P[3275]{
   GP1:
	UF : 7, UT : 3,	CONFIG : 'F U T, 0, 0, 0',
	X =   113.261  mm,	Y =   245.596  mm,	Z =     0.000  mm,
	W =  -167.372 deg,	P =     0.001 deg,	R =   170.283 deg
};
P[3276]{
   GP1:
	UF : 7, UT : 3,	CONFIG : 'F U T, 0, 0, 0',
	X =    97.796  mm,	Y =   252.151  mm,	Z =     0.000  mm,
	W =  -167.372 deg,	P =     0.002 deg,	R =   173.834 deg
};
P[3277]{
   GP1:
	UF : 7, UT : 3,	CONFIG : 'F U T, 0, 0, 0',
	X =    82.004  mm,	Y =   257.731  mm,	Z =     0.000  mm,
	W =  -167.372 deg,	P =     0.002 deg,	R =   177.394 deg
};
P[3278]{
   GP1:
	UF : 7, UT : 3,	CONFIG : 'F U T, 0, 0, 0',
	X =    65.894  mm,	Y =   262.305  mm,	Z =     0.000  mm,
	W =  -167.373 deg,	P =     0.002 deg,	R =  -179.039 deg
};
P[3279]{
   GP1:
	UF : 7, UT : 3,	CONFIG : 'F U T, 0, 0, 0',
	X =    49.508  mm,	Y =   265.883  mm,	Z =     0.000  mm,
	W =  -167.373 deg,	P =     0.003 deg,	R =  -175.483 deg
};
P[3280]{
   GP1:
	UF : 7, UT : 3,	CONFIG : 'F U T, 0, 0, 0',
	X =    31.091  mm,	Y =   268.658  mm,	Z =     0.000  mm,
	W =  -167.374 deg,	P =     0.002 deg,	R =  -171.534 deg
};
P[3281]{
   GP1:
	UF : 7, UT : 3,	CONFIG : 'F U T, 0, 0, 0',
	X =    12.506  mm,	Y =   270.169  mm,	Z =     0.000  mm,
	W =  -167.375 deg,	P =     0.002 deg,	R =  -167.587 deg
};
P[3282]{
   GP1:
	UF : 7, UT : 3,	CONFIG : 'F U T, 0, 0, 0',
	X =    -6.154  mm,	Y =   270.389  mm,	Z =     0.000  mm,
	W =  -167.376 deg,	P =     0.002 deg,	R =  -163.644 deg
};
P[3283]{
   GP1:
	UF : 7, UT : 3,	CONFIG : 'F U T, 0, 0, 0',
	X =   -24.761  mm,	Y =   269.316  mm,	Z =     0.000  mm,
	W =  -167.378 deg,	P =     0.002 deg,	R =  -159.696 deg
};
P[3284]{
   GP1:
	UF : 7, UT : 3,	CONFIG : 'F U T, 0, 0, 0',
	X =   -43.257  mm,	Y =   266.970  mm,	Z =     0.001  mm,
	W =  -167.379 deg,	P =     0.003 deg,	R =  -155.752 deg
};
P[3285]{
   GP1:
	UF : 7, UT : 3,	CONFIG : 'F U T, 0, 0, 0',
	X =   -61.499  mm,	Y =   263.371  mm,	Z =     0.001  mm,
	W =  -167.380 deg,	P =     0.003 deg,	R =  -151.798 deg
};
P[3286]{
   GP1:
	UF : 7, UT : 3,	CONFIG : 'F U T, 0, 0, 0',
	X =   -79.618  mm,	Y =   258.468  mm,	Z =     0.001  mm,
	W =  -167.381 deg,	P =     0.004 deg,	R =  -147.874 deg
};
P[3287]{
   GP1:
	UF : 7, UT : 3,	CONFIG : 'F U T, 0, 0, 0',
	X =   -97.038  mm,	Y =   252.440  mm,	Z =     0.001  mm,
	W =  -167.382 deg,	P =     0.005 deg,	R =  -143.885 deg
};
P[3288]{
   GP1:
	UF : 7, UT : 3,	CONFIG : 'F U T, 0, 0, 0',
	X =  -114.677  mm,	Y =   244.936  mm,	Z =     0.001  mm,
	W =  -167.408 deg,	P =     0.006 deg,	R =  -139.842 deg
};
P[3289]{
   GP1:
	UF : 7, UT : 3,	CONFIG : 'F U T, 0, 0, 0',
	X =  -131.731  mm,	Y =   236.210  mm,	Z =     0.002  mm,
	W =  -167.433 deg,	P =     0.011 deg,	R =  -135.796 deg
};
P[3290]{
   GP1:
	UF : 7, UT : 3,	CONFIG : 'F U T, 0, 0, 0',
	X =  -148.114  mm,	Y =   226.293  mm,	Z =     0.004  mm,
	W =  -167.458 deg,	P =     0.020 deg,	R =  -131.751 deg
};
P[3291]{
   GP1:
	UF : 7, UT : 3,	CONFIG : 'F U T, 0, 0, 0',
	X =  -163.472  mm,	Y =   215.453  mm,	Z =     0.005  mm,
	W =  -167.481 deg,	P =     0.025 deg,	R =  -127.777 deg
};
P[3292]{
   GP1:
	UF : 7, UT : 3,	CONFIG : 'F U T, 0, 0, 0',
	X =  -178.023  mm,	Y =   203.595  mm,	Z =     0.006  mm,
	W =  -167.504 deg,	P =     0.033 deg,	R =  -123.798 deg
};
P[3293]{
   GP1:
	UF : 7, UT : 3,	CONFIG : 'F U T, 0, 0, 0',
	X =  -191.688  mm,	Y =   190.790  mm,	Z =     0.006  mm,
	W =  -167.526 deg,	P =     0.044 deg,	R =  -119.808 deg
};
P[3294]{
   GP1:
	UF : 7, UT : 3,	CONFIG : 'F U T, 0, 0, 0',
	X =  -204.774  mm,	Y =   176.683  mm,	Z =     0.006  mm,
	W =  -167.541 deg,	P =     0.044 deg,	R =  -115.747 deg
};
P[3295]{
   GP1:
	UF : 7, UT : 3,	CONFIG : 'F U T, 0, 0, 0',
	X =  -216.777  mm,	Y =   161.719  mm,	Z =     0.008  mm,
	W =  -167.558 deg,	P =     0.045 deg,	R =  -111.674 deg
};
P[3296]{
   GP1:
	UF : 7, UT : 3,	CONFIG : 'F U T, 0, 0, 0',
	X =  -225.174  mm,	Y =   149.804  mm,	Z =     0.010  mm,
	W =  -167.643 deg,	P =     0.062 deg,	R =  -108.594 deg
};
P[3297]{
   GP1:
	UF : 7, UT : 3,	CONFIG : 'F U T, 0, 0, 0',
	X =  -232.907  mm,	Y =   137.493  mm,	Z =     0.013  mm,
	W =  -167.727 deg,	P =     0.088 deg,	R =  -105.506 deg
};
P[3298]{
   GP1:
	UF : 7, UT : 3,	CONFIG : 'F U T, 0, 0, 0',
	X =  -241.378  mm,	Y =   121.986  mm,	Z =     0.013  mm,
	W =  -167.738 deg,	P =     0.109 deg,	R =  -101.745 deg
};
P[3299]{
   GP1:
	UF : 7, UT : 3,	CONFIG : 'F U T, 0, 0, 0',
	X =  -246.047  mm,	Y =   112.277  mm,	Z =     0.010  mm,
	W =  -167.645 deg,	P =     0.094 deg,	R =   -99.466 deg
};
P[3300]{
   GP1:
	UF : 7, UT : 3,	CONFIG : 'F U T, 0, 0, 0',
	X =  -250.344  mm,	Y =   102.328  mm,	Z =     0.007  mm,
	W =  -167.553 deg,	P =     0.072 deg,	R =   -97.201 deg
};
P[3301]{
   GP1:
	UF : 7, UT : 3,	CONFIG : 'F U T, 0, 0, 0',
	X =  -254.770  mm,	Y =    90.746  mm,	Z =     0.004  mm,
	W =  -167.477 deg,	P =     0.047 deg,	R =   -94.570 deg
};
P[3302]{
   GP1:
	UF : 7, UT : 3,	CONFIG : 'F U T, 0, 0, 0',
	X =  -258.636  mm,	Y =    79.060  mm,	Z =     0.002  mm,
	W =  -167.404 deg,	P =     0.016 deg,	R =   -91.920 deg
};
P[3303]{
   GP1:
	UF : 7, UT : 3,	CONFIG : 'F U T, 0, 0, 0',
	X =  -263.697  mm,	Y =    60.088  mm,	Z =     0.001  mm,
	W =  -167.393 deg,	P =     0.014 deg,	R =   -87.773 deg
};
P[3304]{
   GP1:
	UF : 7, UT : 3,	CONFIG : 'F U T, 0, 1, 0',
	X =  -267.363  mm,	Y =    40.814  mm,	Z =     0.000  mm,
	W =  -167.383 deg,	P =     0.011 deg,	R =   -83.624 deg
};
P[3305]{
   GP1:
	UF : 7, UT : 3,	CONFIG : 'F U T, 0, 1, 0',
	X =  -269.616  mm,	Y =    21.277  mm,	Z =     0.000  mm,
	W =  -167.373 deg,	P =     0.007 deg,	R =   -79.483 deg
};
P[3306]{
   GP1:
	UF : 7, UT : 3,	CONFIG : 'F U T, 0, 1, 0',
	X =  -270.465  mm,	Y =     0.000  mm,	Z =     0.000  mm,
	W =  -167.363 deg,	P =     0.001 deg,	R =   -75.503 deg
};
P[3307]{
   GP1:
	UF : 7, UT : 3,	CONFIG : 'F U T, 0, 1, 0',
	X =  -270.465  mm,	Y =     0.000  mm,	Z =     0.000  mm,
	W =  -167.363 deg,	P =     0.001 deg,	R =   -75.503 deg
};
P[3308]{
   GP1:
	UF : 7, UT : 3,	CONFIG : 'F U T, 0, 1, 0',
	X =  -270.465  mm,	Y =     0.000  mm,	Z =     0.000  mm,
	W =  -167.363 deg,	P =     0.001 deg,	R =   -75.503 deg
};
P[3309]{
   GP1:
	UF : 7, UT : 3,	CONFIG : 'F U T, 0, 1, 0',
	X =  -270.465  mm,	Y =     0.000  mm,	Z =     0.000  mm,
	W =  -167.363 deg,	P =     0.001 deg,	R =   -75.503 deg
};
P[3310]{
   GP1:
	UF : 7, UT : 3,
	J1 =  -129.583 deg,	J2 =    24.319 deg,	J3 =   -28.425 deg,
	J4 =   110.695 deg,	J5 =   124.219 deg,	J6 =   -55.036 deg
};
/END
